PROGRAM MAIN
VAR
	fbnci :FB_NCI;
	
	stChannelInput  AT %I*: NCTOPLC_NCICHANNEL_REF;
	stChannelOutput AT %Q*: PLCTONC_NCICHANNEL_REF;


END_VAR


X_Axis();
Y_Axis();
Z_Axis();
PANEL();

fbnci(
	sProgramName:='mdi_2.nc' , 
	stChannelInput:=stChannelInput , 
	stChannelOutput:=stChannelOutput , 
	stAxRefAxX:=gvl.Axis_X , 
	stAxRefAyY:=gvl.Axis_Y );

END_PROGRAM

(* stored: Version 1.1.0.1, ProductVersion 3.1.4024.13
   POU MAIN: Id {71784bf4-c468-4ab3-a04c-eac2f366ca9b}, SpecialFunc None *)
